% RSLogix 500 project LIMO_WEST_BIN_WASH_FEB_9_2022_10_57_AM_BAK012.RSS, saved by version 11.00.00.00 %
PROJECT "JBT BIN"    % processor: MicroLogix 1200 %

PROGRAM FILES
  LAD 2   8 rungs
  LAD 3   3 rungs
  LAD 4   11 rungs
  LAD 5   29 rungs
  LAD 6   9 rungs
  LAD 7   11 rungs
  LAD 8   7 rungs
  LAD 9   27 rungs

DATA FILES
  O0 OUTPUT  4 elements
  I1 INPUT  4 elements
  S2 STATUS  66 elements
  B3 BINARY  4 elements
  T4 TIMER  18 elements
  C5 COUNTER  1 elements
  R6 CONTROL  1 elements
  N7 INTEGER  6 elements
  F8 FLOAT  1 elements
  L9   1 elements
  L10   2 elements

LADDER 2
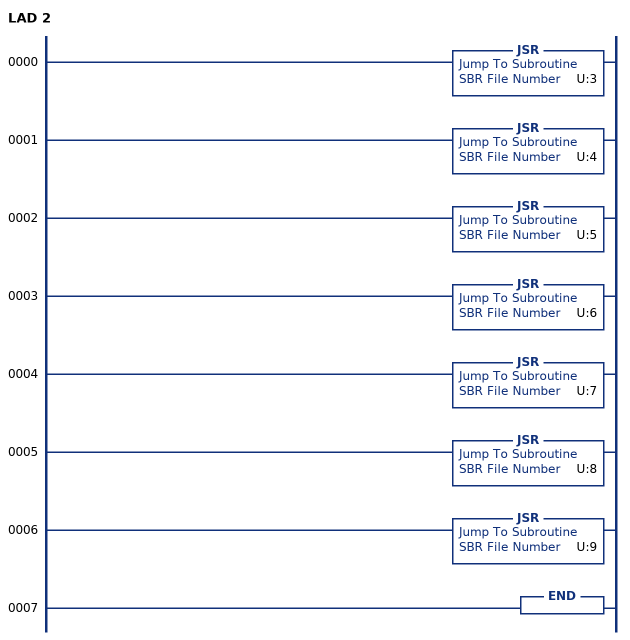
% Rung: 0 %
SOR JSR U:3 EOR
% Rung: 1 %
SOR JSR U:4 EOR
% Rung: 2 %
SOR JSR U:5 EOR
% Rung: 3 %
SOR JSR U:6 EOR
% Rung: 4 %
SOR JSR U:7 EOR
% Rung: 5 %
SOR JSR U:8 EOR
% Rung: 6 %
SOR JSR U:9 EOR
% Rung: 7 %
SOR END EOR

LADDER 3
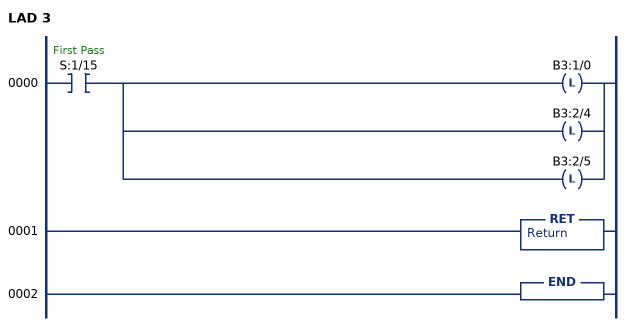
% Rung: 0 %
SOR XIC S:1/15 BST OTL B3:1/0 NXB BST OTL B3:2/4 NXB OTL B3:2/5 BND BND EOR
%   S:1/15  "First Pass" %
% Rung: 1 %
SOR RET EOR
% Rung: 2 %
SOR END EOR

LADDER 4
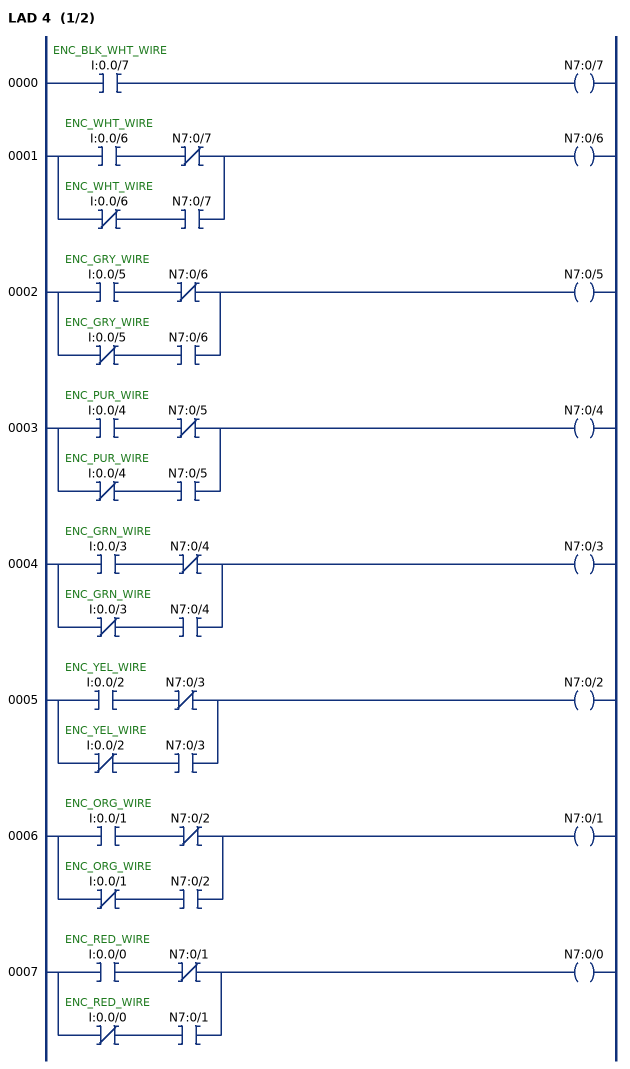
% Rung: 0 %
SOR XIC I:0.0/7 OTE N7:0/7 EOR
%   I:0.0/7  ENC_BLK_WHT_WIRE %
% Rung: 1 %
SOR BST XIC I:0.0/6 XIO N7:0/7 NXB XIO I:0.0/6 XIC N7:0/7 BND OTE N7:0/6 EOR
%   I:0.0/6  ENC_WHT_WIRE %
% Rung: 2 %
SOR BST XIC I:0.0/5 XIO N7:0/6 NXB XIO I:0.0/5 XIC N7:0/6 BND OTE N7:0/5 EOR
%   I:0.0/5  ENC_GRY_WIRE %
% Rung: 3 %
SOR BST XIC I:0.0/4 XIO N7:0/5 NXB XIO I:0.0/4 XIC N7:0/5 BND OTE N7:0/4 EOR
%   I:0.0/4  ENC_PUR_WIRE %
% Rung: 4 %
SOR BST XIC I:0.0/3 XIO N7:0/4 NXB XIO I:0.0/3 XIC N7:0/4 BND OTE N7:0/3 EOR
%   I:0.0/3  ENC_GRN_WIRE %
% Rung: 5 %
SOR BST XIC I:0.0/2 XIO N7:0/3 NXB XIO I:0.0/2 XIC N7:0/3 BND OTE N7:0/2 EOR
%   I:0.0/2  ENC_YEL_WIRE %
% Rung: 6 %
SOR BST XIC I:0.0/1 XIO N7:0/2 NXB XIO I:0.0/1 XIC N7:0/2 BND OTE N7:0/1 EOR
%   I:0.0/1  ENC_ORG_WIRE %
% Rung: 7 %
SOR BST XIC I:0.0/0 XIO N7:0/1 NXB XIO I:0.0/0 XIC N7:0/1 BND OTE N7:0/0 EOR
%   I:0.0/0  ENC_RED_WIRE %

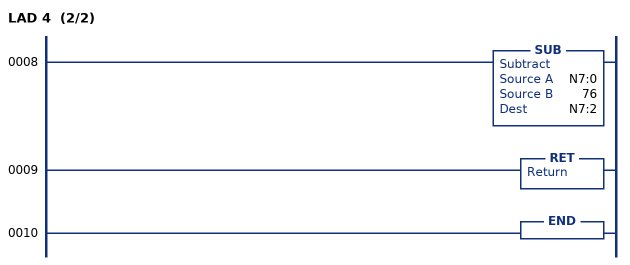
% Rung: 8 %
SOR SUB N7:0 76 N7:2 EOR
% Rung: 9 %
SOR RET EOR
% Rung: 10 %
SOR END EOR

LADDER 5
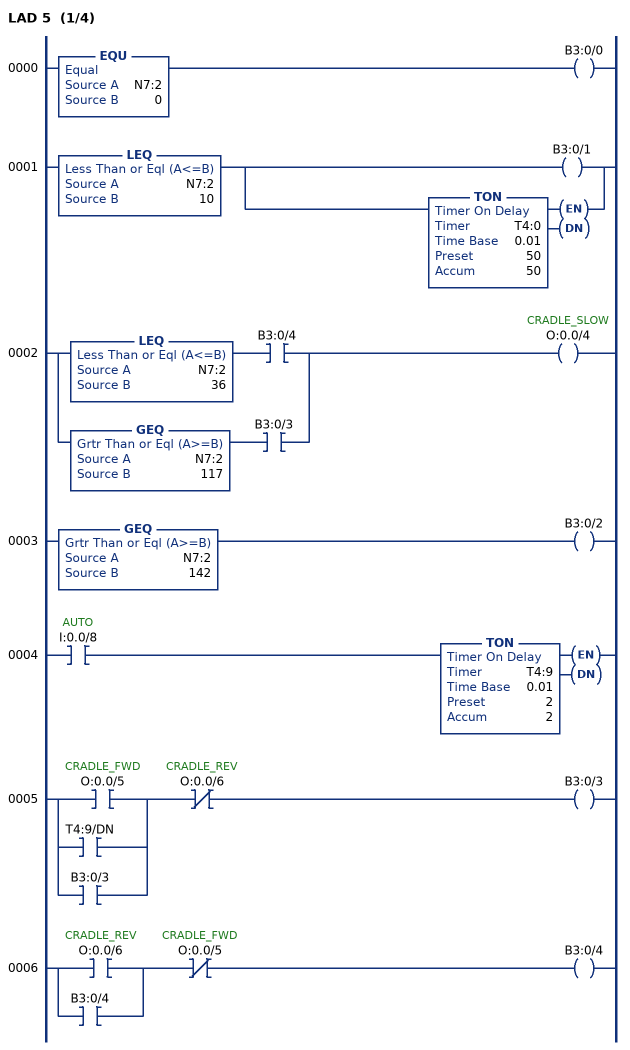
% Rung: 0 %
SOR EQU N7:2 0 OTE B3:0/0 EOR
% Rung: 1 %
SOR LEQ N7:2 10 BST OTE B3:0/1 NXB TON T4:0 0.01 50 50 BND EOR
% Rung: 2 %
SOR BST LEQ N7:2 36 XIC B3:0/4 NXB GEQ N7:2 117 XIC B3:0/3 BND OTE O:0.0/4 EOR
%   O:0.0/4  CRADLE_SLOW %
% Rung: 3 %
SOR GEQ N7:2 142 OTE B3:0/2 EOR
% Rung: 4 %
SOR XIC I:0.0/8 TON T4:9 0.01 2 2 EOR
%   I:0.0/8  AUTO %
% Rung: 5 %
SOR BST XIC O:0.0/5 NXB XIC T4:9/DN NXB XIC B3:0/3 BND XIO O:0.0/6 OTE B3:0/3 EOR
%   O:0.0/5  CRADLE_FWD %
%   O:0.0/6  CRADLE_REV %
% Rung: 6 %
SOR BST XIC O:0.0/6 NXB XIC B3:0/4 BND XIO O:0.0/5 OTE B3:0/4 EOR
%   O:0.0/6  CRADLE_REV %
%   O:0.0/5  CRADLE_FWD %

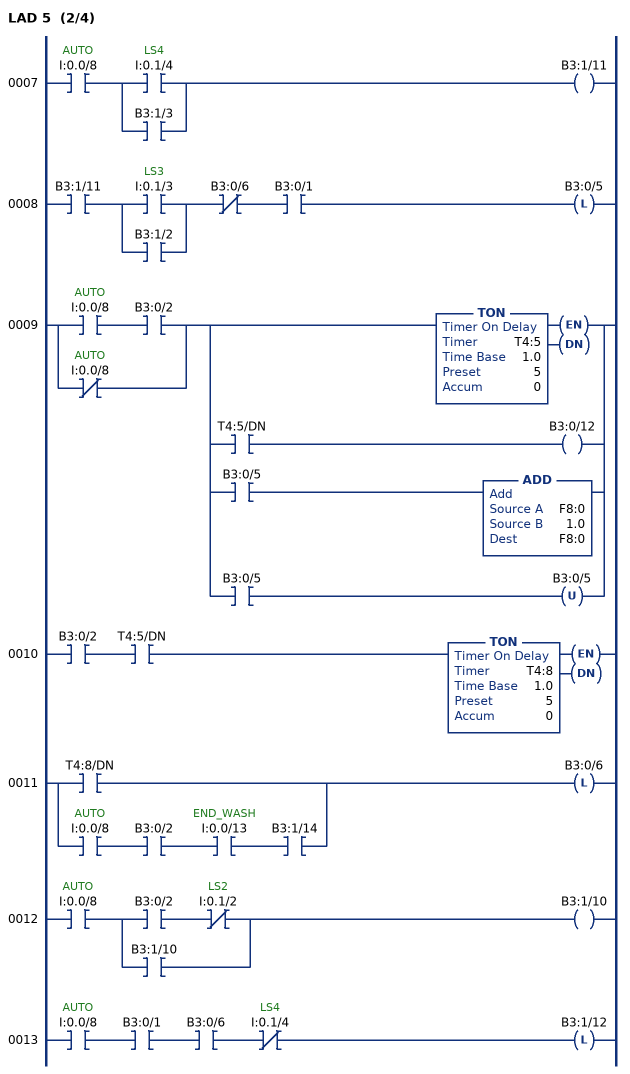
% Rung: 7 %
SOR XIC I:0.0/8 BST XIC I:0.1/4 NXB XIC B3:1/3 BND OTE B3:1/11 EOR
%   I:0.0/8  AUTO %
%   I:0.1/4  LS4 %
% Rung: 8 %
SOR XIC B3:1/11 BST XIC I:0.1/3 NXB XIC B3:1/2 BND XIO B3:0/6 XIC B3:0/1 OTL B3:0/5 EOR
%   I:0.1/3  LS3 %
% Rung: 9 %
SOR BST XIC I:0.0/8 XIC B3:0/2 NXB XIO I:0.0/8 BND BST TON T4:5 1.0 5 0 NXB XIC T4:5/DN OTE B3:0/12 NXB BST XIC B3:0/5 ADD F8:0 1.0 F8:0 NXB XIC B3:0/5 OTU B3:0/5 BND BND EOR
%   I:0.0/8  AUTO %
% Rung: 10 %
SOR XIC B3:0/2 XIC T4:5/DN TON T4:8 1.0 5 0 EOR
% Rung: 11 %
SOR BST XIC T4:8/DN NXB XIC I:0.0/8 XIC B3:0/2 XIC I:0.0/13 XIC B3:1/14 BND OTL B3:0/6 EOR
%   I:0.0/8  AUTO %
%   I:0.0/13  END_WASH %
% Rung: 12 %
SOR XIC I:0.0/8 BST XIC B3:0/2 XIO I:0.1/2 NXB XIC B3:1/10 BND OTE B3:1/10 EOR
%   I:0.0/8  AUTO %
%   I:0.1/2  LS2 %
% Rung: 13 %
SOR XIC I:0.0/8 XIC B3:0/1 XIC B3:0/6 XIO I:0.1/4 OTL B3:1/12 EOR
%   I:0.0/8  AUTO %
%   I:0.1/4  LS4 %

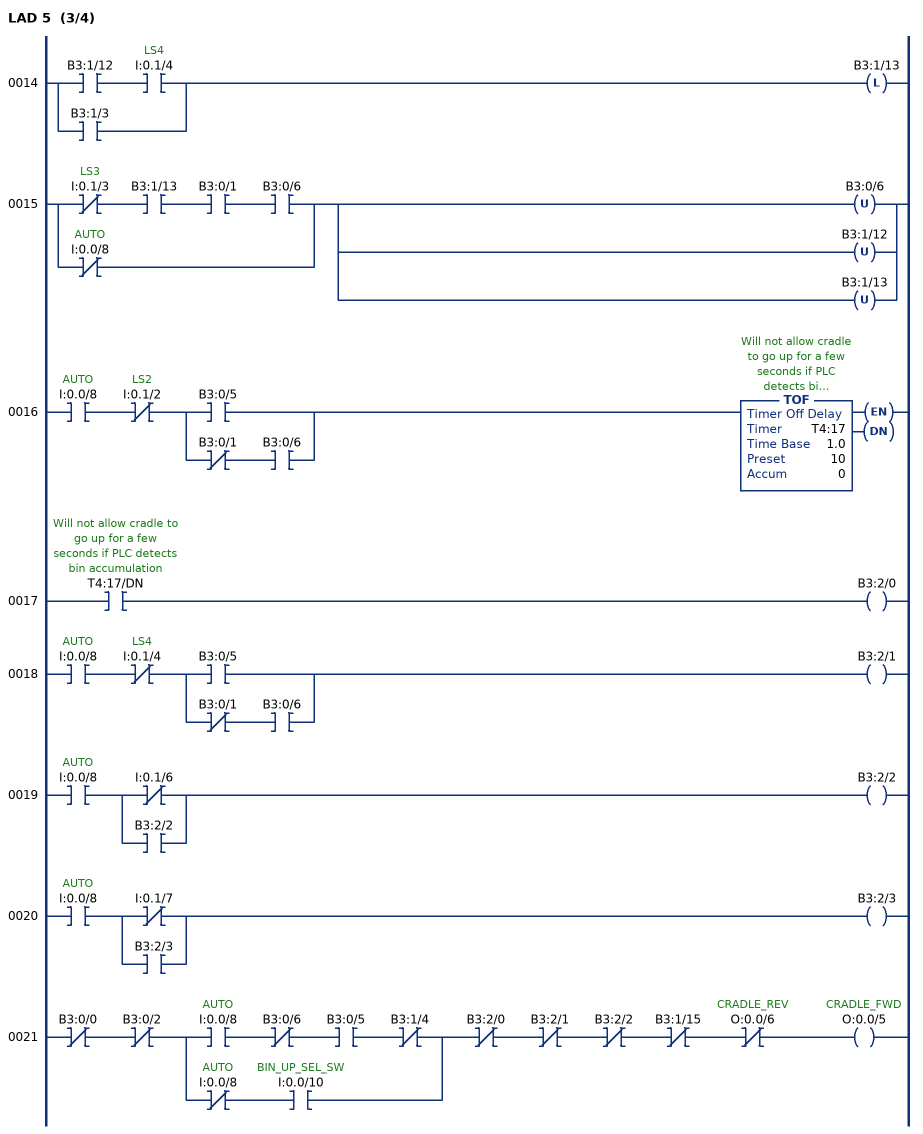
% Rung: 14 %
SOR BST XIC B3:1/12 XIC I:0.1/4 NXB XIC B3:1/3 BND OTL B3:1/13 EOR
%   I:0.1/4  LS4 %
% Rung: 15 %
SOR BST XIO I:0.1/3 XIC B3:1/13 XIC B3:0/1 XIC B3:0/6 NXB XIO I:0.0/8 BND BST OTU B3:0/6 NXB BST OTU B3:1/12 NXB OTU B3:1/13 BND BND EOR
%   I:0.1/3  LS3 %
%   I:0.0/8  AUTO %
% Rung: 16 %
SOR XIC I:0.0/8 XIO I:0.1/2 BST XIC B3:0/5 NXB XIO B3:0/1 XIC B3:0/6 BND TOF T4:17 1.0 10 0 EOR
%   I:0.0/8  AUTO %
%   I:0.1/2  LS2 %
%   T4:17  "Will not allow cradle to go up for a few seconds if PLC detects bin accumulation" %
% Rung: 17 %
SOR XIC T4:17/DN OTE B3:2/0 EOR
%   T4:17  "Will not allow cradle to go up for a few seconds if PLC detects bin accumulation" %
% Rung: 18 %
SOR XIC I:0.0/8 XIO I:0.1/4 BST XIC B3:0/5 NXB XIO B3:0/1 XIC B3:0/6 BND OTE B3:2/1 EOR
%   I:0.0/8  AUTO %
%   I:0.1/4  LS4 %
% Rung: 19 %
SOR XIC I:0.0/8 BST XIO I:0.1/6 NXB XIC B3:2/2 BND OTE B3:2/2 EOR
%   I:0.0/8  AUTO %
% Rung: 20 %
SOR XIC I:0.0/8 BST XIO I:0.1/7 NXB XIC B3:2/3 BND OTE B3:2/3 EOR
%   I:0.0/8  AUTO %
% Rung: 21 %
SOR XIO B3:0/0 XIO B3:0/2 BST XIC I:0.0/8 XIO B3:0/6 XIC B3:0/5 XIO B3:1/4 NXB XIO I:0.0/8 XIC I:0.0/10 BND XIO B3:2/0 XIO B3:2/1 XIO B3:2/2 XIO B3:1/15 XIO O:0.0/6 OTE O:0.0/5 EOR
%   I:0.0/8  AUTO %
%   I:0.0/10  BIN_UP_SEL_SW %
%   O:0.0/6  CRADLE_REV %
%   O:0.0/5  CRADLE_FWD %

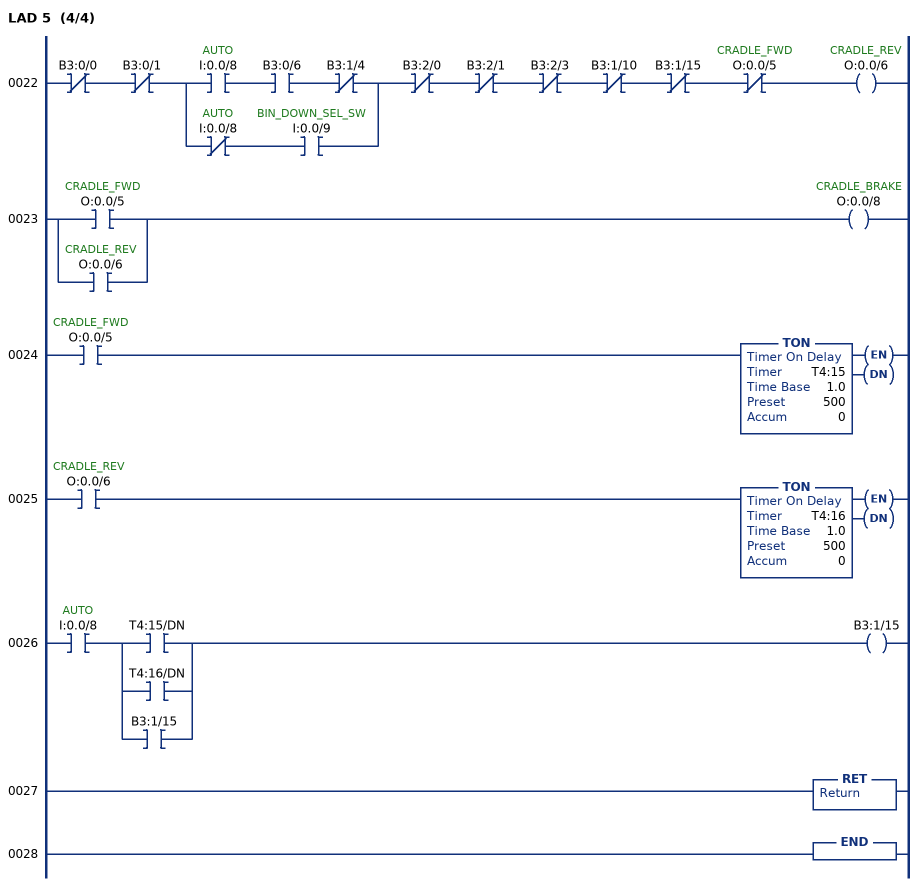
% Rung: 22 %
SOR XIO B3:0/0 XIO B3:0/1 BST XIC I:0.0/8 XIC B3:0/6 XIO B3:1/4 NXB XIO I:0.0/8 XIC I:0.0/9 BND XIO B3:2/0 XIO B3:2/1 XIO B3:2/3 XIO B3:1/10 XIO B3:1/15 XIO O:0.0/5 OTE O:0.0/6 EOR
%   I:0.0/8  AUTO %
%   I:0.0/9  BIN_DOWN_SEL_SW %
%   O:0.0/5  CRADLE_FWD %
%   O:0.0/6  CRADLE_REV %
% Rung: 23 %
SOR BST XIC O:0.0/5 NXB XIC O:0.0/6 BND OTE O:0.0/8 EOR
%   O:0.0/5  CRADLE_FWD %
%   O:0.0/6  CRADLE_REV %
%   O:0.0/8  CRADLE_BRAKE %
% Rung: 24 %
SOR XIC O:0.0/5 TON T4:15 1.0 500 0 EOR
%   O:0.0/5  CRADLE_FWD %
% Rung: 25 %
SOR XIC O:0.0/6 TON T4:16 1.0 500 0 EOR
%   O:0.0/6  CRADLE_REV %
% Rung: 26 %
SOR XIC I:0.0/8 BST BST XIC T4:15/DN NXB XIC T4:16/DN BND NXB XIC B3:1/15 BND OTE B3:1/15 EOR
%   I:0.0/8  AUTO %
% Rung: 27 %
SOR RET EOR
% Rung: 28 %
SOR END EOR

LADDER 6
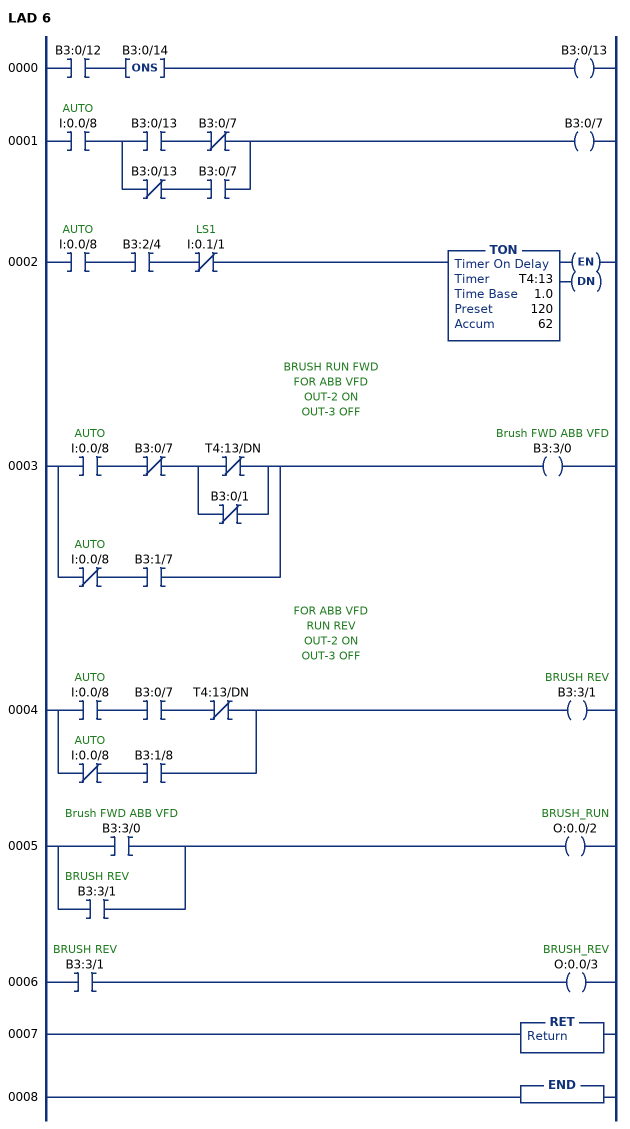
% Rung: 0 %
SOR XIC B3:0/12 ONS B3:0/14 OTE B3:0/13 EOR
% Rung: 1 %
SOR XIC I:0.0/8 BST XIC B3:0/13 XIO B3:0/7 NXB XIO B3:0/13 XIC B3:0/7 BND OTE B3:0/7 EOR
%   I:0.0/8  AUTO %
% Rung: 2 %
SOR XIC I:0.0/8 XIC B3:2/4 XIO I:0.1/1 TON T4:13 1.0 120 62 EOR
%   I:0.0/8  AUTO %
%   I:0.1/1  LS1 %
% Rung: 3 %
% BRUSH RUN FWD
% 
% FOR ABB VFD
% OUT-2 ON
% OUT-3 OFF %
SOR BST XIC I:0.0/8 XIO B3:0/7 BST XIO T4:13/DN NXB XIO B3:0/1 BND NXB XIO I:0.0/8 XIC B3:1/7 BND OTE B3:3/0 EOR
%   I:0.0/8  AUTO %
%   B3:3/0  "Brush FWD ABB VFD" %
% Rung: 4 %
% FOR ABB VFD
% RUN REV
% OUT-2 ON
% OUT-3 OFF %
SOR BST XIC I:0.0/8 XIC B3:0/7 XIO T4:13/DN NXB XIO I:0.0/8 XIC B3:1/8 BND OTE B3:3/1 EOR
%   I:0.0/8  AUTO %
%   B3:3/1  "BRUSH REV" %
% Rung: 5 %
SOR BST XIC B3:3/0 NXB XIC B3:3/1 BND OTE O:0.0/2 EOR
%   B3:3/0  "Brush FWD ABB VFD" %
%   B3:3/1  "BRUSH REV" %
%   O:0.0/2  BRUSH_RUN %
% Rung: 6 %
SOR XIC B3:3/1 OTE O:0.0/3 EOR
%   B3:3/1  "BRUSH REV" %
%   O:0.0/3  BRUSH_REV %
% Rung: 7 %
SOR RET EOR
% Rung: 8 %
SOR END EOR

LADDER 7
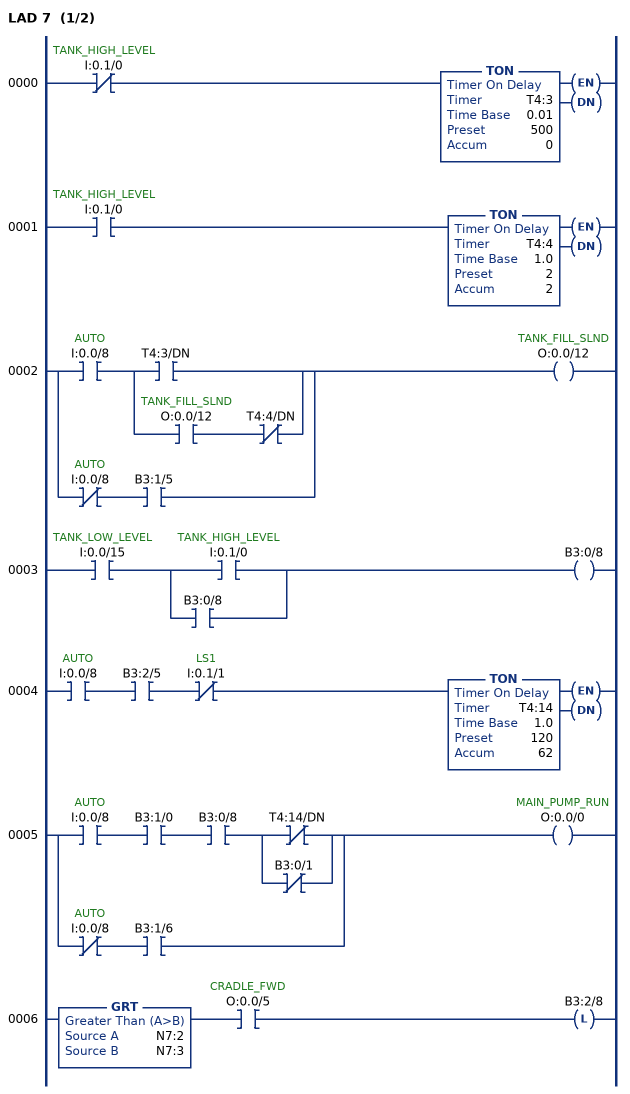
% Rung: 0 %
SOR XIO I:0.1/0 TON T4:3 0.01 500 0 EOR
%   I:0.1/0  TANK_HIGH_LEVEL %
% Rung: 1 %
SOR XIC I:0.1/0 TON T4:4 1.0 2 2 EOR
%   I:0.1/0  TANK_HIGH_LEVEL %
% Rung: 2 %
SOR BST XIC I:0.0/8 BST XIC T4:3/DN NXB XIC O:0.0/12 XIO T4:4/DN BND NXB XIO I:0.0/8 XIC B3:1/5 BND OTE O:0.0/12 EOR
%   I:0.0/8  AUTO %
%   O:0.0/12  TANK_FILL_SLND %
% Rung: 3 %
SOR XIC I:0.0/15 BST XIC I:0.1/0 NXB XIC B3:0/8 BND OTE B3:0/8 EOR
%   I:0.0/15  TANK_LOW_LEVEL %
%   I:0.1/0  TANK_HIGH_LEVEL %
% Rung: 4 %
SOR XIC I:0.0/8 XIC B3:2/5 XIO I:0.1/1 TON T4:14 1.0 120 62 EOR
%   I:0.0/8  AUTO %
%   I:0.1/1  LS1 %
% Rung: 5 %
SOR BST XIC I:0.0/8 XIC B3:1/0 XIC B3:0/8 BST XIO T4:14/DN NXB XIO B3:0/1 BND NXB XIO I:0.0/8 XIC B3:1/6 BND OTE O:0.0/0 EOR
%   I:0.0/8  AUTO %
%   O:0.0/0  MAIN_PUMP_RUN %
% Rung: 6 %
SOR GRT N7:2 N7:3 XIC O:0.0/5 OTL B3:2/8 EOR
%   O:0.0/5  CRADLE_FWD %

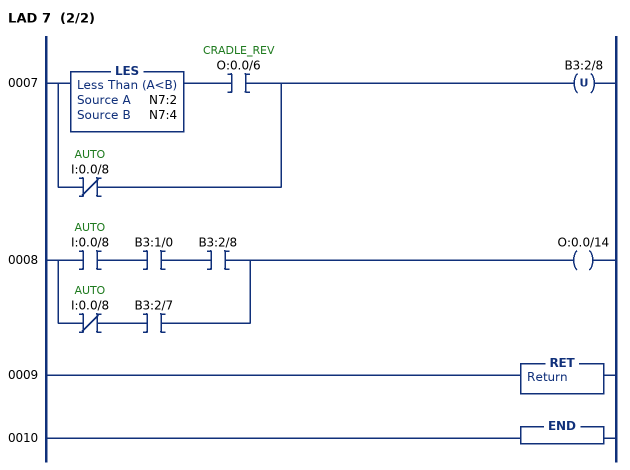
% Rung: 7 %
SOR BST LES N7:2 N7:4 XIC O:0.0/6 NXB XIO I:0.0/8 BND OTU B3:2/8 EOR
%   O:0.0/6  CRADLE_REV %
%   I:0.0/8  AUTO %
% Rung: 8 %
SOR BST XIC I:0.0/8 XIC B3:1/0 XIC B3:2/8 NXB XIO I:0.0/8 XIC B3:2/7 BND OTE O:0.0/14 EOR
%   I:0.0/8  AUTO %
% Rung: 9 %
SOR RET EOR
% Rung: 10 %
SOR END EOR

LADDER 8
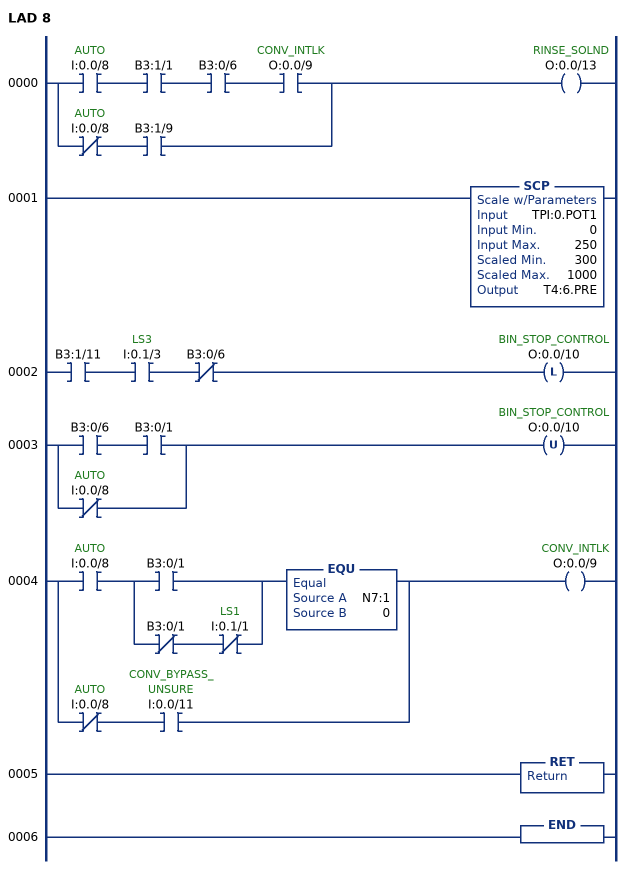
% Rung: 0 %
SOR BST XIC I:0.0/8 XIC B3:1/1 XIC B3:0/6 XIC O:0.0/9 NXB XIO I:0.0/8 XIC B3:1/9 BND OTE O:0.0/13 EOR
%   I:0.0/8  AUTO %
%   O:0.0/9  CONV_INTLK %
%   O:0.0/13  RINSE_SOLND %
% Rung: 1 %
SOR SCP TPI:0.POT1 0 250 300 1000 T4:6.PRE EOR
% Rung: 2 %
SOR XIC B3:1/11 XIC I:0.1/3 XIO B3:0/6 OTL O:0.0/10 EOR
%   I:0.1/3  LS3 %
%   O:0.0/10  BIN_STOP_CONTROL %
% Rung: 3 %
SOR BST XIC B3:0/6 XIC B3:0/1 NXB XIO I:0.0/8 BND OTU O:0.0/10 EOR
%   I:0.0/8  AUTO %
%   O:0.0/10  BIN_STOP_CONTROL %
% Rung: 4 %
SOR BST XIC I:0.0/8 BST XIC B3:0/1 NXB XIO B3:0/1 XIO I:0.1/1 BND EQU N7:1 0 NXB XIO I:0.0/8 XIC I:0.0/11 BND OTE O:0.0/9 EOR
%   I:0.0/8  AUTO %
%   I:0.1/1  LS1 %
%   I:0.0/11  CONV_BYPASS_UNSURE %
%   O:0.0/9  CONV_INTLK %
% Rung: 5 %
SOR RET EOR
% Rung: 6 %
SOR END EOR

LADDER 9
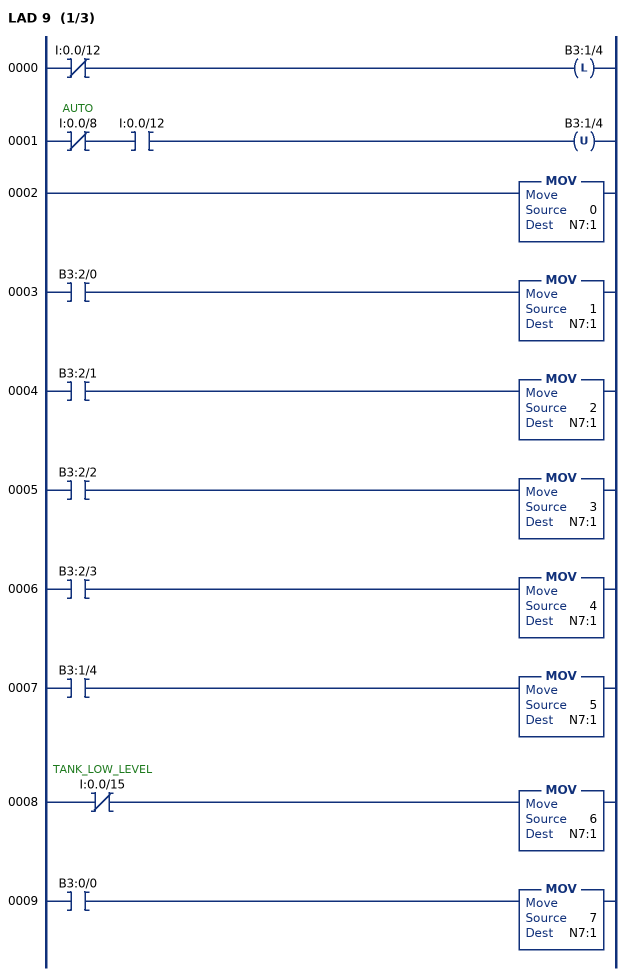
% Rung: 0 %
SOR XIO I:0.0/12 OTL B3:1/4 EOR
% Rung: 1 %
SOR XIO I:0.0/8 XIC I:0.0/12 OTU B3:1/4 EOR
%   I:0.0/8  AUTO %
% Rung: 2 %
SOR MOV 0 N7:1 EOR
% Rung: 3 %
SOR XIC B3:2/0 MOV 1 N7:1 EOR
% Rung: 4 %
SOR XIC B3:2/1 MOV 2 N7:1 EOR
% Rung: 5 %
SOR XIC B3:2/2 MOV 3 N7:1 EOR
% Rung: 6 %
SOR XIC B3:2/3 MOV 4 N7:1 EOR
% Rung: 7 %
SOR XIC B3:1/4 MOV 5 N7:1 EOR
% Rung: 8 %
SOR XIO I:0.0/15 MOV 6 N7:1 EOR
%   I:0.0/15  TANK_LOW_LEVEL %
% Rung: 9 %
SOR XIC B3:0/0 MOV 7 N7:1 EOR

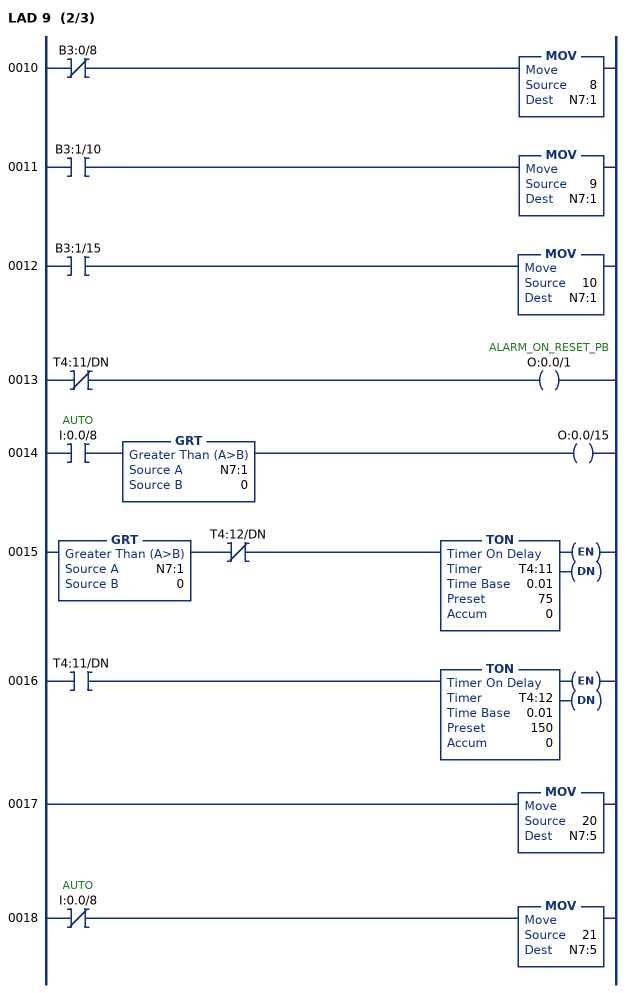
% Rung: 10 %
SOR XIO B3:0/8 MOV 8 N7:1 EOR
% Rung: 11 %
SOR XIC B3:1/10 MOV 9 N7:1 EOR
% Rung: 12 %
SOR XIC B3:1/15 MOV 10 N7:1 EOR
% Rung: 13 %
SOR XIO T4:11/DN OTE O:0.0/1 EOR
%   O:0.0/1  ALARM_ON_RESET_PB %
% Rung: 14 %
SOR XIC I:0.0/8 GRT N7:1 0 OTE O:0.0/15 EOR
%   I:0.0/8  AUTO %
% Rung: 15 %
SOR GRT N7:1 0 XIO T4:12/DN TON T4:11 0.01 75 0 EOR
% Rung: 16 %
SOR XIC T4:11/DN TON T4:12 0.01 150 0 EOR
% Rung: 17 %
SOR MOV 20 N7:5 EOR
% Rung: 18 %
SOR XIO I:0.0/8 MOV 21 N7:5 EOR
%   I:0.0/8  AUTO %

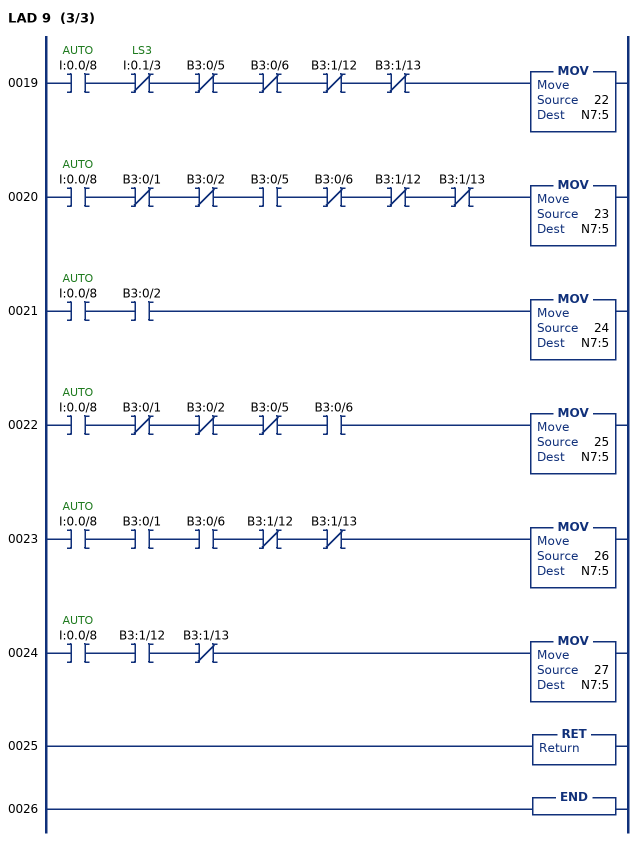
% Rung: 19 %
SOR XIC I:0.0/8 XIO I:0.1/3 XIO B3:0/5 XIO B3:0/6 XIO B3:1/12 XIO B3:1/13 MOV 22 N7:5 EOR
%   I:0.0/8  AUTO %
%   I:0.1/3  LS3 %
% Rung: 20 %
SOR XIC I:0.0/8 XIO B3:0/1 XIO B3:0/2 XIC B3:0/5 XIO B3:0/6 XIO B3:1/12 XIO B3:1/13 MOV 23 N7:5 EOR
%   I:0.0/8  AUTO %
% Rung: 21 %
SOR XIC I:0.0/8 XIC B3:0/2 MOV 24 N7:5 EOR
%   I:0.0/8  AUTO %
% Rung: 22 %
SOR XIC I:0.0/8 XIO B3:0/1 XIO B3:0/2 XIO B3:0/5 XIC B3:0/6 MOV 25 N7:5 EOR
%   I:0.0/8  AUTO %
% Rung: 23 %
SOR XIC I:0.0/8 XIC B3:0/1 XIC B3:0/6 XIO B3:1/12 XIO B3:1/13 MOV 26 N7:5 EOR
%   I:0.0/8  AUTO %
% Rung: 24 %
SOR XIC I:0.0/8 XIC B3:1/12 XIO B3:1/13 MOV 27 N7:5 EOR
%   I:0.0/8  AUTO %
% Rung: 25 %
SOR RET EOR
% Rung: 26 %
SOR END EOR

OTHER DOCUMENTED ADDRESSES
  T0:17  "safety timer"

DATA TABLE (non-zero values as saved)
DATA B3
% B3:0 % 0X0DDA 0X4A03 0X8030 0X0000
DATA T4
% .PRE .ACC %
% T4:0 % 50 50
% T4:1 % 1 0
% T4:2 % 1 0
% T4:3 % 500 0
% T4:4 % 2 2
% T4:5 % 5 0
% T4:6 % 681 0
% T4:7 % 375 500
% T4:8 % 5 0
% T4:9 % 2 2
% T4:10 % 500 0
% T4:11 % 75 0
% T4:12 % 150 0
% T4:13 % 120 62
% T4:14 % 120 62
% T4:15 % 500 0
% T4:16 % 500 0
% T4:17 % 10 0
DATA N7
% N7:0 % 84 0 8 65 130 26
DATA F8
% F8:0 % 240270
